// TIA Portal V16 export
// export: Created 2023-06-21T17:06:29.2417224Z, ExportSetting WithDefaults, DisplayName Totally Integrated Automation Portal, DisplayVersion V16 Update 4, DisplayName TIA Portal Version Control Interface, DisplayVersion V16 Update 2, DisplayName TIA Portal Openness, DisplayVersion V16 Update 4, DisplayName SINAMICS Startdrive Advanced, DisplayVersion V16, DisplayName SINAMICS Startdrive G130, G150, S120, S150, SINAMICS MV, S210, DisplayVersion V16, DisplayName SINAMICS Startdrive G110M, G120, G120C, G120D, G120P, DisplayVersion V16, DisplayName STEP 7 Professional, DisplayVersion V16 Update 4, DisplayName STEP 7 Safety, DisplayVersion V16, DisplayName Soft Starter ES, DisplayVersion V16, DisplayName WinCC Advanced, DisplayVersion V16 Update 4
DATA_BLOCK "Modbus_Send_Receive_1"   // DB13
{ S7_Optimized_Access := 'FALSE' }
VERSION : 0.1
// stored: AutoNumber false, DBAccessibleFromOPCUA true, IsOnlyStoredInLoadMemory false, IsWriteProtectedInAS false
   VAR
      Reading_Struct : Struct
         "32001" : Word;   // STS_UNIT_01
         "32002" : Word;   // OPER_UNIT_01
         "32003" : Word;   // SP_UNIT_01
         "32004" : Word;   // ERROR_UNIT_01
         "32005" : Word;   // PV_UNIT_01
         "32006" : Word;   // SERROR_UNIT_01
         "32007" : Word;   // STS_UNIT_02
         "32008" : Word;   // OPER_UNIT_02
         "32009" : Word;   // SP_UNIT_02
         "32010" : Word;   // ERROR_UNIT_02
         "32011" : Word;   // PV_UNIT_02
         "32012" : Word;   // SERROR_UNIT_02
         "32013" : Word;   // STS_UNIT_01
         "32014" : Word;   // OPER_UNIT_01
         "32015" : Word;   // SP_UNIT_01
         "32016" : Word;   // ERROR_UNIT_01
         "32017" : Word;   // PV_UNIT_01
         "32018" : Word;   // SERROR_UNIT_01
         "32019" : Word;   // STS_UNIT_02
         "32020" : Word;   // OPER_UNIT_02
         "32021" : Word;   // SP_UNIT_02
         "32022" : Word;   // ERROR_UNIT_02
         "32023" : Word;   // PV_UNIT_02
         "32024" : Word;   // SERROR_UNIT_02
         "32025" : Word;   // STS_UNIT_01
         "32026" : Word;   // OPER_UNIT_01
         "32027" : Word;   // SP_UNIT_01
         "32028" : Word;   // ERROR_UNIT_01
         "32029" : Word;   // PV_UNIT_01
         "32030" : Word;   // SERROR_UNIT_01
         "32031" : Word;   // STS_UNIT_02
         "32032" : Word;   // OPER_UNIT_02
         "32033" : Word;   // SP_UNIT_02
         "32034" : Word;   // ERROR_UNIT_02
         "32035" : Word;   // PV_UNIT_02
         "32036" : Word;   // SERROR_UNIT_02
         "32037" : Word;   // STS_UNIT_01
         "32038" : Word;   // OPER_UNIT_01
         "32039" : Word;   // SP_UNIT_01
         "32040" : Word;   // ERROR_UNIT_01
         "32041" : Word;   // PV_UNIT_01
         "32042" : Word;   // SERROR_UNIT_01
         "32043" : Word;   // STS_UNIT_02
         "32044" : Word;   // OPER_UNIT_02
         "32045" : Word;   // SP_UNIT_02
         "32046" : Word;   // ERROR_UNIT_02
         "32047" : Word;   // PV_UNIT_02
         "32048" : Word;   // SERROR_UNIT_02
         "32049" : Word;   // STS_UNIT_01
         "32050" : Word;   // OPER_UNIT_01
         "32051" : Word;   // SP_UNIT_01
         "32052" : Word;   // ERROR_UNIT_01
         "32053" : Word;   // PV_UNIT_01
         "32054" : Word;   // SERROR_UNIT_01
         "32055" : Word;   // STS_UNIT_02
         "32056" : Word;   // OPER_UNIT_02
         "32057" : Word;   // SP_UNIT_02
         "32058" : Word;   // ERROR_UNIT_02
         "32059" : Word;   // PV_UNIT_02
         "32060" : Word;   // SERROR_UNIT_02
         "32061" : Word;   // STS_UNIT_01
         "32062" : Word;   // OPER_UNIT_01
         "32063" : Word;   // SP_UNIT_01
         "32064" : Word;   // ERROR_UNIT_01
         "32065" : Word;   // PV_UNIT_01
         "32066" : Word;   // SERROR_UNIT_01
         "32067" : Word;   // STS_UNIT_02
         "32068" : Word;   // OPER_UNIT_02
         "32069" : Word;   // SP_UNIT_02
         "32070" : Word;   // ERROR_UNIT_02
         "32071" : Word;   // PV_UNIT_02
         "32072" : Word;   // SERROR_UNIT_02
         "32073" : Word;   // STS_UNIT_01
         "32074" : Word;   // OPER_UNIT_01
         "32075" : Word;   // SP_UNIT_01
         "32076" : Word;   // ERROR_UNIT_01
         "32077" : Word;   // PV_UNIT_01
         "32078" : Word;   // SERROR_UNIT_01
         "32079" : Word;   // STS_UNIT_02
         "32080" : Word;   // OPER_UNIT_02
         "32081" : Word;   // SP_UNIT_02
         "32082" : Word;   // ERROR_UNIT_02
         "32083" : Word;   // PV_UNIT_02
         "32084" : Word;   // SERROR_UNIT_02
         "40001" : Word;
         "42001" : Word;   // STS
         "42002" : Word;   // OPER_MODE
         "42003" : Word;   // SP
         "42004" : Word;
         "42005" : Word;
         "42006" : Word;
         "42007" : Word;
         "42008" : Word;
         "42009" : Word;
         "42010" : Word;
         "42011" : Word;
         "42012" : Word;
         "42013" : Word;
         "42014" : Word;
         "42015" : Word;
         "42016" : Word;
         "42017" : Word;
         "42018" : Word;
         "42019" : Word;
         "42020" : Word;
         "42021" : Word;
         "42022" : Word;
         "42023" : Word;
         "42024" : Word;
         "42025" : Word;
         "42026" : Word;
         "42027" : Word;
         "42028" : Word;
         "42029" : Word;
         "42030" : Word;
         "42031" : Word;
         "42032" : Word;
         "42033" : Word;
         "42034" : Word;
         "42035" : Word;
         "42036" : Word;
         "42037" : Word;
         "42038" : Word;
         "42039" : Word;
         "42040" : Word;
         "42041" : Word;
         "42042" : Word;
      END_STRUCT;
      Reading_Struct_2 : Struct
         "30001" : Word;
         "30002" : Word;   // COMM_OK = 3FFF
      END_STRUCT;
      Extrusora_1 : Struct
         Ligado : Bool;
         Fan : Bool;
         Heating : Bool;
         Cooling : Bool;
         Sts_Fan : Bool;
         Sts_Heating : Bool;
         Sts_Cooling : Bool;
         Slave : Bool;
         Master : Bool;
         SP : Word;
         PV : Word;
      END_STRUCT;
      Extrusora_2 : Struct
         Ligado : Bool;
         Fan : Bool;
         Heating : Bool;
         Cooling : Bool;
         Sts_Fan : Bool;
         Sts_Heating : Bool;
         Sts_Cooling : Bool;
         Slave : Bool;
         Master : Bool;
         SP : Word;
         PV : Word;
      END_STRUCT;
      Extrusora_3 : Struct
         Ligado : Bool;
         Fan : Bool;
         Heating : Bool;
         Cooling : Bool;
         Sts_Fan : Bool;
         Sts_Heating : Bool;
         Sts_Cooling : Bool;
         Slave : Bool;
         Master : Bool;
         SP : Word;
         PV : Word;
      END_STRUCT;
      Extrusora_4 : Struct
         Ligado : Bool;
         Fan : Bool;
         Heating : Bool;
         Cooling : Bool;
         Sts_Fan : Bool;
         Sts_Heating : Bool;
         Sts_Cooling : Bool;
         Slave : Bool;
         Master : Bool;
         SP : Word;
         PV : Word;
      END_STRUCT;
      Extrusora_5 : Struct
         Ligado : Bool;
         Fan : Bool;
         Heating : Bool;
         Cooling : Bool;
         Sts_Fan : Bool;
         Sts_Heating : Bool;
         Sts_Cooling : Bool;
         Slave : Bool;
         Master : Bool;
         SP : Word;
         PV : Word;
      END_STRUCT;
      Extrusora_6 : Struct
         Ligado : Bool;
         Fan : Bool;
         Heating : Bool;
         Cooling : Bool;
         Sts_Fan : Bool;
         Sts_Heating : Bool;
         Sts_Cooling : Bool;
         Slave : Bool;
         Master : Bool;
         SP : Word;
         PV : Word;
      END_STRUCT;
      Extrusora_7 : Struct
         Ligado : Bool;
         Fan : Bool;
         Heating : Bool;
         Cooling : Bool;
         Sts_Fan : Bool;
         Sts_Heating : Bool;
         Sts_Cooling : Bool;
         Slave : Bool;
         Master : Bool;
         SP : Word;
         PV : Word;
      END_STRUCT;
      Extrusora_8 : Struct
         Ligado : Bool;
         Fan : Bool;
         Heating : Bool;
         Cooling : Bool;
         Sts_Fan : Bool;
         Sts_Heating : Bool;
         Sts_Cooling : Bool;
         Slave : Bool;
         Master : Bool;
         SP : Word;
         PV : Word;
      END_STRUCT;
      Extrusora_9 : Struct
         Ligado : Bool;
         Fan : Bool;
         Heating : Bool;
         Cooling : Bool;
         Sts_Fan : Bool;
         Sts_Heating : Bool;
         Sts_Cooling : Bool;
         Slave : Bool;
         Master : Bool;
         SP : Word;
         PV : Word;
      END_STRUCT;
      Extrusora_10 : Struct
         Ligado : Bool;
         Fan : Bool;
         Heating : Bool;
         Cooling : Bool;
         Sts_Fan : Bool;
         Sts_Heating : Bool;
         Sts_Cooling : Bool;
         Slave : Bool;
         Master : Bool;
         SP : Word;
         PV : Word;
      END_STRUCT;
      Extrusora_11 : Struct
         Ligado : Bool;
         Fan : Bool;
         Heating : Bool;
         Cooling : Bool;
         Sts_Fan : Bool;
         Sts_Heating : Bool;
         Sts_Cooling : Bool;
         Slave : Bool;
         Master : Bool;
         SP : Word;
         PV : Word;
      END_STRUCT;
      Extrusora_12 : Struct
         Ligado : Bool;
         Fan : Bool;
         Heating : Bool;
         Cooling : Bool;
         Sts_Fan : Bool;
         Sts_Heating : Bool;
         Sts_Cooling : Bool;
         Slave : Bool;
         Master : Bool;
         SP : Word;
         PV : Word;
      END_STRUCT;
      Extrusora_13 : Struct
         Ligado : Bool;
         Fan : Bool;
         Heating : Bool;
         Cooling : Bool;
         Sts_Fan : Bool;
         Sts_Heating : Bool;
         Sts_Cooling : Bool;
         Slave : Bool;
         Master : Bool;
         SP : Word;
         PV : Word;
      END_STRUCT;
      Extrusora_14 : Struct
         Ligado : Bool;
         Fan : Bool;
         Heating : Bool;
         Cooling : Bool;
         Sts_Fan : Bool;
         Sts_Heating : Bool;
         Sts_Cooling : Bool;
         Slave : Bool;
         Master : Bool;
         SP : Word;
         PV : Word;
      END_STRUCT;
      Malfunction_1 : Bool;
      Malfunction_2 : Bool;
      Malfunction_3 : Bool;
      Malfunction_4 : Bool;
      Malfunction_5 : Bool;
      Malfunction_6 : Bool;
      Malfunction_7 : Bool;
      Malfunction_8 : Bool;
      Malfunction_9 : Bool;
      Malfunction_10 : Bool;
      Malfunction_11 : Bool;
      Malfunction_12 : Bool;
      Malfunction_13 : Bool;
      Malfunction_14 : Bool;
   END_VAR
BEGIN
END_DATA_BLOCK
